INTERFACE I_Datatypes EXTENDS I_EventEmitter

METHOD PUBLIC Accept
VAR_INPUT
	Visitor : I_DatatypeVisitor;
END_VAR
END_METHOD

METHOD RegisterDatatype
VAR_INPUT
	Datatype : I_Datatype;
END_VAR
END_METHOD

METHOD PUBLIC SerializeTypeWith
VAR_INPUT
	Serializer : I_Serializer;
END_VAR
END_METHOD

METHOD PUBLIC TryGetAliasByIdentifier : BOOL
VAR_INPUT
	Identifier : T_MAXSTRING;
	Destination : REFERENCE TO I_AliasDatatype;
END_VAR
END_METHOD

METHOD PUBLIC TryGetArrayByIdentifier : BOOL
VAR_INPUT
	Identifier : T_MAXSTRING;
	Destination : REFERENCE TO I_ArrayDatatype;
END_VAR
END_METHOD

METHOD PUBLIC TryGetEnumByIdentifier : BOOL
VAR_INPUT
	Identifier : T_MAXSTRING;
	Destination : REFERENCE TO I_EnumDatatype;
END_VAR
END_METHOD

METHOD PUBLIC TryGetInterfaceByIdentifier : BOOL
VAR_INPUT
	Identifier : T_MAXSTRING;
	Destination : REFERENCE TO I_InterfaceDatatype;
END_VAR
END_METHOD

METHOD PUBLIC TryGetPrimitiveByTypeName : BOOL
VAR_INPUT
	TypeName : T_MAXSTRING;
	Destination : REFERENCE TO I_AliasDatatype;
END_VAR
END_METHOD

METHOD PUBLIC TryGetStructureByIdentifier : BOOL
VAR_INPUT
	Identifier : T_MAXSTRING;
	Destination : REFERENCE TO I_StructuredDatatype;
END_VAR
END_METHOD

END_INTERFACE

(* stored: Version 1.1.0.1, ProductVersion 3.1.4024.13
   Itf I_Datatypes: Id {fa5985fa-0352-0837-008f-2100e7182f33}
   Method Accept: Id {ab5a6019-b90b-0356-36ad-ac3b7614d57c}
   Method RegisterDatatype: Id {a28830d7-6191-0883-0e41-e4c205ba804e}
   Method SerializeTypeWith: Id {13366319-95e0-0db8-0311-946242514cd9}
   Method TryGetAliasByIdentifier: Id {2eb48292-09ae-0ce3-2529-21e731dfd8cb}
   Method TryGetArrayByIdentifier: Id {1e77a6ee-f035-0aa3-0935-9ed4ab35e6a3}
   Method TryGetEnumByIdentifier: Id {cc8c44b8-14d0-0287-11a5-56136f79c410}
   Method TryGetInterfaceByIdentifier: Id {1987a886-9c50-0c24-3782-dd3c813dde2b}
   Method TryGetPrimitiveByTypeName: Id {84f9f9c9-5063-0c47-1c42-af2f88c84dd0}
   Method TryGetStructureByIdentifier: Id {4071e151-c73c-0bed-3454-9ed0692110c3} *)
